RoboDK station: Conveying-Decanting-and-Material-Handling-with-Fanuc-R-2000iC-165F.rdk

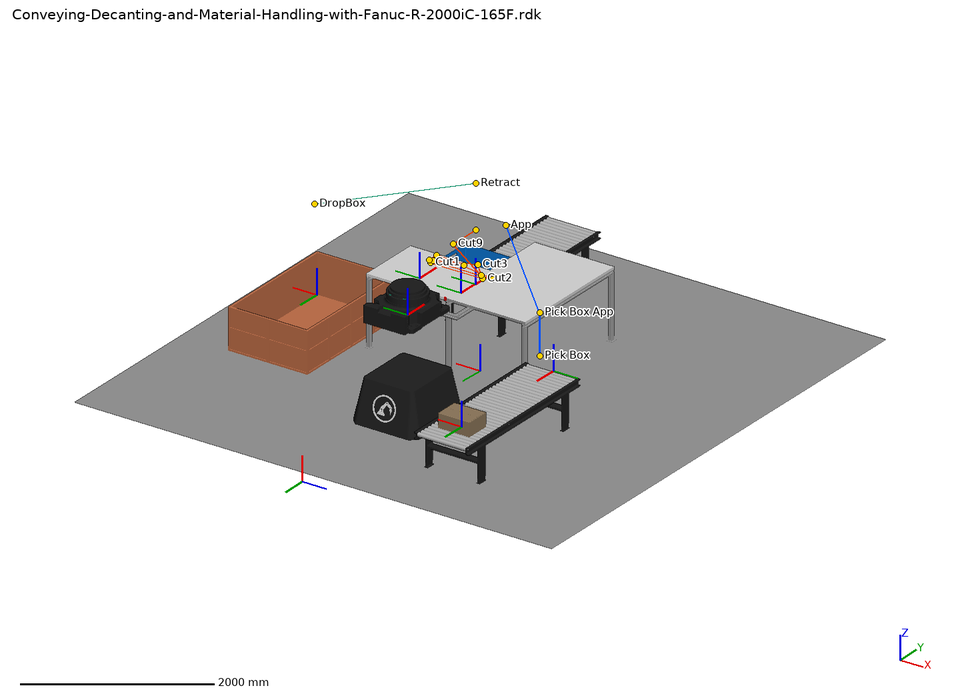
[picture v0: the station drawn from its stored meshes, robots at their saved joint values, targets as dots, program paths as lines]
Station Conveying, Decanting and Material Handling with Fanuc R-2000iC/165F (saved by RoboDK 5.9.2). Poses are relative to the parent item; angles as X-Y-Z fixed-axis rotations.
Station parameters (name, value as stored): TAGS, ['Decanting']
  - frame Roller Conveyor In Base at (1190, -380, 485) mm, rotated rx 0 ry 0 rz -90 deg
    - robot Roller Conveyor In: 1 axes
        modified DH rows (alpha deg, a mm, theta deg, d mm): 0, 0, 0, 0 linear
        base shift (0, 0, -485) mm, rotated rx 0 ry 90 rz 0 deg
        joint limits [-20000] to [20000]; home [0]; saved at [1400]
      - frame Conveyor In Ref at (230, -10, 5) mm, rotated rx 0 ry 0 rz -90 deg
        - frame BoxRef at (0, 0, 0) mm
          - object Decanting Box Bottom at (0, 0, 0) mm, size 400 x 300 x 6 mm, geometry from Decanting Box v4.step
          - object Decanting Box Top at (0, 0, 0) mm, size 400 x 300 x 166 mm, geometry from Decanting Box v4.step
          - object RoboDK_logo at (135, -20, 160) mm, rotated rx 0 ry 0 rz 90 deg, size 280 x 130 x 161.8 mm
          - object RoboDK_logo at (5, -20, 160) mm, rotated rx 0 ry 0 rz 90 deg, size 280 x 130 x 161.8 mm
          - object RoboDK_logo at (-125, -20, 160) mm, rotated rx 0 ry 0 rz 90 deg, size 280 x 130 x 161.8 mm
    - target Conv In 1 (Cartesian target) at (1400, 0, 0) mm; joints [1400, -18.458, 3.617, 0, -93.617, -148.241] of Roller Conveyor In
    - target Conv In 2 (Cartesian target) at (0, 0, 0) mm; joints [0, -18.458, 3.617, 0, -93.617, -148.241] of Roller Conveyor In
  - frame Roller Conveyor Out Base at (-640, 570, 485) mm, rotated rx 0 ry 0 rz 90 deg
    - robot Roller Conveyor Out: 1 axes
        modified DH rows (alpha deg, a mm, theta deg, d mm): 0, 0, 0, 0 linear
        base shift (0, 0, -485) mm, rotated rx 0 ry 90 rz 0 deg
        joint limits [-20000] to [20000]; home [0]; saved at [0]
      - frame Conveyor Out Ref at (250, -10, 0) mm
        - object Caisse Modulaire at (0, 0, 0) mm, size 460 x 580 x 300 mm, geometry from Caisse Modulaire v5.step
  - frame Gravity Base at (0, 0, 0) mm, rotated rx 0 ry 0 rz 180 deg
    - robot Gravity: 1 axes
        modified DH rows (alpha deg, a mm, theta deg, d mm): 0, 0, 0, 0 linear
        joint limits [0] to [900000]; home [0]; saved at [0]
      - frame GravityRef at (0, 3190, 0) mm
      - tool Gravity TCP, TCP at (0, 0, 0) mm
    - target BoxDrop1 (Cartesian target) at (0, 0, -355) mm, rotated rx 0 ry -90 rz 0 deg; joints [355, 40.194, -30.706, 0, -59.294, 73.523] of Gravity
    - target BoxDrop2 (Cartesian target) at (0, 0, -1505) mm, rotated rx 0 ry -90 rz 0 deg; joints [1505, 40.194, -30.706, 0, -59.294, 73.523] of Gravity
  - frame Fanuc R-2000iC/165F Base at (0, -1300, 1160) mm, rotated rx 0 ry 0 rz 90 deg
    - robot Fanuc R-2000iC/165F: 6 axes, payload 165 kg, reach 2655 mm, repeatability 0.2 mm, weight 1170 kg
        joint limits [-185, -56, -65, -360, -125, -360] to [185, 80, 245, 360, 125, 360]; home [0, 0, 0, 0, 0, 0]; saved at [5.758, -15.413, -35.804, 0, -54.196, -95.758]
      - tool Decanting gripper v3, TCP at (0, 0, 200) mm, size 405 x 200 x 270 mm, geometry from Decanting gripper v3.step
      - frame BoxOpening Base at (0, -148, 458) mm
        - robot BoxOpening: 1 axes
            modified DH rows (alpha deg, a mm, theta deg, d mm): 0, 0, 0, 0
            base shift (0, 0, 0) mm, rotated rx 0 ry 90 rz 0 deg
            joint limits [-360] to [360]; home [0]; saved at [0]
          - tool BoxOpeningTCP, TCP at (0, 0, 0) mm
    - object Pedestal H500mm (Type 2) at (0, 0, -1160) mm, rotated rx 0 ry 0 rz 90 deg, size 844.5 x 933.7 x 500 mm, geometry from Pedestal-H500mm-Type-2.sld
    - target Pick Box (Cartesian target) at (690, -1180, -415) mm, rotated rx -180 ry 0 rz -90 deg; joints [-59.683, 14.803, -63.072, 0, -26.928, -30.317] of Fanuc R-2000iC/165F
    - target Pick Box App (Cartesian target) at (690, -1180, 75) mm, rotated rx -180 ry 0 rz -90 deg; joints [-59.683, -5.784, -36.452, 0, -53.548, -30.317] of Fanuc R-2000iC/165F
    - target App (Cartesian target) at (1570, -140, 435) mm, rotated rx -180 ry 0 rz -90 deg; joints [-5.096, -0.842, -19.934, 0, -70.066, -84.904] of Fanuc R-2000iC/165F
    - frame Table at (1300, 0, -1160) mm, rotated rx 0 ry 0 rz 90 deg
      - object Decanting table assem at (-220, -1380, 485) mm, rotated rx 0 ry 0 rz -180 deg, size 2035.1 x 1855.1 x 855 mm, geometry from Decanting table assem v12.step
      - target Cut1 (Cartesian target) at (570, 70, 1106) mm, rotated rx 180 ry 0 rz -180 deg; joints [24.864, -2.283, -43.25, 0, -46.75, -114.864] of Fanuc R-2000iC/165F
      - target Cut2 (Cartesian target) at (-80, 70, 1106) mm, rotated rx 180 ry 0 rz 180 deg; joints [-3.721, -9.346, -42.545, 0, -47.455, -86.279] of Fanuc R-2000iC/165F
      - target Cut3 (Cartesian target) at (140, -170, 1106) mm, rotated rx 180 ry 0 rz -180 deg; joints [5.44, 4.103, -43.15, 0, -46.85, -95.44] of Fanuc R-2000iC/165F
      - target Cut4 (Cartesian target) at (570, 20, 1106) mm, rotated rx 180 ry 0 rz -90 deg; joints [24.004, 0.173, -43.295, 0, -46.705, -24.004] of Fanuc R-2000iC/165F
      - target Cut5 (Cartesian target) at (-170, 20, 1106) mm, rotated rx -180 ry 0 rz -90 deg; joints [-7.565, -5.895, -42.995, 0, -47.005, 7.565] of Fanuc R-2000iC/165F
      - target Cut6 (Cartesian target) at (620, -110, 1106) mm, rotated rx 180 ry 0 rz 0 deg; joints [23.736, 7.305, -42.836, 0, -47.164, 66.264] of Fanuc R-2000iC/165F
      - target Cut7 (Cartesian target) at (620, 20, 1106) mm, rotated rx 180 ry 0 rz 90 deg; joints [25.844, 1.287, -43.28, 0, -46.72, 154.156] of Fanuc R-2000iC/165F
      - target Cut8 (Cartesian target) at (-30, 20, 1106) mm, rotated rx 180 ry 0 rz 90 deg; joints [-1.343, -6.523, -42.928, 0, -47.072, 181.343] of Fanuc R-2000iC/165F
      - target Cut9 (Cartesian target) at (630, -420, 1106) mm, rotated rx -180 ry 0 rz 0 deg; joints [20.117, 21.228, -39.525, 0, -50.475, 69.883] of Fanuc R-2000iC/165F
      - target Cut10 (Cartesian target) at (630, -830, 1106) mm, rotated rx 180 ry 0 rz 0 deg; joints [16.477, 40.194, -30.706, 0, -59.294, 73.523] of Fanuc R-2000iC/165F
    - target Retract (Cartesian target) at (2130, 630, 476) mm, rotated rx -180 ry 0 rz 90 deg; joints [16.477, 34.546, -9.725, 0, -80.275, 73.523] of Fanuc R-2000iC/165F
    - target DropBox (Cartesian target) at (1120, 1950, 276) mm, rotated rx -180 ry 0 rz 90 deg; joints [60.129, 37.062, -17.345, 0, -72.655, 29.871] of Fanuc R-2000iC/165F
    - target Home (Cartesian target) at (1190, 120, 55) mm, rotated rx 180 ry 0 rz -90 deg; joints [5.758, -15.413, -35.804, 0, -54.196, -95.758] of Fanuc R-2000iC/165F
  - frame Container at (-2400, 500, 0) mm, rotated rx 0 ry 0 rz 180 deg
    - object Container at (0, 0, 0) mm, size 1000 x 1600 x 500 mm, geometry from Container.step
  - object Floor at (0, 0, 0) mm, rotated rx 0 ry 0 rz 180 deg, size 6000 x 6000 x 0 mm, geometry from Floor.sld
  - program Main (19 instructions, listed below)
  - folder Python
    - Python program OpenBox (listed below)
    - Python program MechnaismReset (listed below)
    - Python program ConveyorReset (listed below)
    - Python program SwitchRef_Box_to_convOut (listed below)
  - folder Programs
    - program Gravity_BoxDrop2 (3 instructions, listed below)
    - program CutBox (14 instructions, listed below)
    - program RecycleBox (7 instructions, listed below)
  - program Home (3 instructions, listed below)
  - program Conv In (2 instructions, listed below)
  - program Reset (4 instructions, listed below)
  - notes Description: <!DOCTYPE HTML PUBLIC "-//W3C//DTD HTML 4.0//EN" "http://www.w3.org/TR/REC-html40/strict.dtd">
<html><head><meta name="qrichtext" content="1" /><style type="text/css">
p, li { white-space: pre-wrap; }
</style></head><body style=" font-family:'MS Shell Dlg 2'; font-size:8.25pt; font-weight:400; font-style:normal;">
<p style=" margin-top:0px; margin-bottom:0px; margin-left:0px; margin-right:0px; -qt-block-indent:0; text-indent:0px;">This example demonstrates a box emptying and sorting application using an industrial 6-axis Fanuc R-2000iC/165F robot equipped with a vacuum gripper. The robot picks a closed box from a roller conveyor and opens its bottom by sliding it across a stationary knife mounted on a flat table. It then pushes the opened box toward a bin, allowing the contents to fall out. After emptying, the robot discards the empty box into a designated container.</p></body></html>
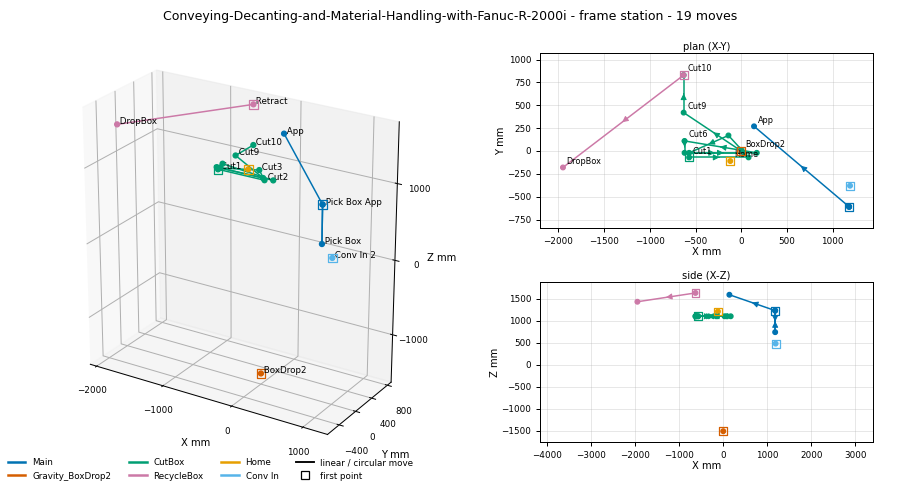
[picture p0: tool path of Conveying-Decanting-and-Material-Handling-with-Fanuc-R-2000iC-165F.rdk in frame station, 19 of 19 moves have a stored position in this frame; points joined in program order, loops and branches not executed]

--- program Main (robot Fanuc R-2000iC/165F) ---
  Call Reset
  Set Ref.: Fanuc R-2000iC/165F Base
  Set Tool: Decanting gripper v3
  Call Home
  Call Conv In
  MoveJ (Pick Box App)
  MoveL (Pick Box)
  Attach to Decanting gripper v3
  Attach to Decanting gripper v3
  Attach to Decanting gripper v3
  Attach to Decanting gripper v3
  Attach to Decanting gripper v3
  MoveL (Pick Box App)
  MoveL (App)
  Call CutBox
  Call OpenBox
  Call SwitchRef_Box_to_convOut
  Call RecycleBox
  Call Home

--- Python program OpenBox ---
# Type help("robodk.robolink") or help("robodk.robomath") for more information
# Press F5 to run the script
# Documentation: https://robodk.com/doc/en/RoboDK-API.html
# Reference:     https://robodk.com/doc/en/PythonAPI/robodk.html
# Note: It is not required to keep a copy of this file, your Python script is saved with your RDK project

# You can also use the new version of the API:
from robodk import robolink    # RoboDK API
from robodk import robomath    # Robot toolbox
import time
RDK = robolink.Robolink()

#----- Constant -----

MECHANISM_NAME1 = 'BoxOpening'
MECHANISM_NAME2 = 'Gravity'
PART_TRAVEL_MM = 0
Target1 = RDK.Item("BoxDrop1")

#Declaration of the frames
frame1 = RDK.Item('Decanting gripper v3')
frame2 = RDK.Item('BoxOpeningTCP')

item1 = RDK.Item("Decanting Box Bottom")
item2 = RDK.Item("RoboDK_logo")

gravityframe = RDK.Item("GravityRef")

#Declaration of the child frames
obj_list1 = frame1.Childs()
obj_list2 = frame2.Childs()

mechanism1 = RDK.Item(MECHANISM_NAME1)
mechanism2 = RDK.Item(MECHANISM_NAME2)

if mechanism1.Valid():
  mechanism1.MoveJ([0])

#open box
for item in obj_list1:
  if item.Name() == item1.Name():
      item.setParentStatic(frame2)

if mechanism1.Valid():
  mechanism1.MoveJ([90])

for item in obj_list2:
    item.setParentStatic(frame1)

#drop box
for item in obj_list1:
  if item.Name() == item1.Name():
    item.setParentStatic(frame2)

#Gravity
for item in obj_list1:
  if item.Name() == item2.Name():
    item.setParentStatic(gravityframe)

if mechanism2.Valid():
  mechanism2.setJoints([0])
  mechanism2.MoveL(Target1)

--- Python program MechnaismReset ---
# Type help("robodk.robolink") or help("robodk.robomath") for more information
# Press F5 to run the script
# Documentation: https://robodk.com/doc/en/RoboDK-API.html
# Reference:     https://robodk.com/doc/en/PythonAPI/robodk.html
# Note: It is not required to keep a copy of this file, your Python script is saved with your RDK project

# You can also use the new version of the API:
from robodk import robolink    # RoboDK API
from robodk import robomath    # Robot toolbox
RDK = robolink.Robolink()

#----- Constant -----

MECHANISM_NAME1 = 'BoxOpening'
MECHANISM_NAME2 = 'Gravity'

mechanism1 = RDK.Item(MECHANISM_NAME1)
mechanism2 = RDK.Item(MECHANISM_NAME2)

if mechanism1.Valid():
  mechanism1.setJoints([0])

if mechanism2.Valid():
  mechanism2.setJoints([0])

--- Python program ConveyorReset ---
# Type help("robodk.robolink") or help("robodk.robomath") for more information
# Press F5 to run the script
# Documentation: https://robodk.com/doc/en/RoboDK-API.html
# Reference:     https://robodk.com/doc/en/PythonAPI/robodk.html
# Note: It is not required to keep a copy of this file, your Python script is saved with your RDK project

# You can also use the new version of the API:
from robodk import robolink    # RoboDK API
from robodk import robomath    # Robot toolbox
RDK = robolink.Robolink()

#----- Constant -----
MECHANISM_NAME1 = 'Roller Conveyor In'#Name of the conveyor mechanism
MECHANISM_NAME2 = 'Roller Conveyor Out'#Name of the conveyor mechanism
MECHANISM_NAME3 = 'Gravity'#Name of the conveyor mechanism
PART_TRAVEL_MM = 0 #Travel for each box

mechanism1 = RDK.Item(MECHANISM_NAME1)
if mechanism1.Valid():
    mechanism1.setJoints([1400.00])

mechanism2 = RDK.Item(MECHANISM_NAME2)
if mechanism2.Valid():
    mechanism2.setJoints([0])


mechanism3 = RDK.Item(MECHANISM_NAME3)
if mechanism3.Valid():
    mechanism3.setJoints([0])

--- Python program SwitchRef_Box_to_convOut ---
# Type help("robodk.robolink") or help("robodk.robomath") for more information
# Press F5 to run the script
# Documentation: https://robodk.com/doc/en/RoboDK-API.html
# Reference:     https://robodk.com/doc/en/PythonAPI/robodk.html
# Note: It is not required to keep a copy of this file, your Python script is saved with your RDK project

# You can also use the new version of the API:
from robodk import robolink    # RoboDK API
from robodk import robomath    # Robot toolbox
import time
RDK = robolink.Robolink()

#----- Constant -----
Target1 = RDK.Item("BoxDrop1")

#Declaration of the frames
frame3 = RDK.Item("Conveyor Out Ref")

item1 = RDK.Item("Decanting Box Bottom")
item2 = RDK.Item("RoboDK_logo")

gravityframe = RDK.Item("GravityRef")

#Declaration of the child frames
obj_list4 = gravityframe.Childs()

#Switch to conveyor ref
for item in obj_list4:
    item.setParentStatic(frame3)

--- program Gravity_BoxDrop2 (robot Gravity) ---
  Set Ref.: Gravity Base
  Set Tool: Gravity TCP
  MoveL (BoxDrop2)

--- program CutBox (robot Fanuc R-2000iC/165F) ---
  Set Ref.: Table
  Set Tool: Decanting gripper v3
  Set speed (200.0 mm/s)
  MoveL (Cut1)
  MoveL (Cut2)
  MoveL (Cut3)
  MoveL (Cut4)
  MoveL (Cut5)
  MoveL (Cut6)
  MoveL (Cut7)
  MoveL (Cut8)
  MoveL (Cut9)
  MoveL (Cut10)
  Set speed (600.0 mm/s)

--- program RecycleBox (robot Fanuc R-2000iC/165F) ---
  Set Ref.: Fanuc R-2000iC/165F Base
  Set Tool: Decanting gripper v3
  MoveL (Retract)
  MoveL (DropBox)
  Detach from Decanting gripper v3
  Detach from BoxOpeningTCP
  Call Gravity_BoxDrop2

--- program Home (robot Fanuc R-2000iC/165F) ---
  Set Ref.: Fanuc R-2000iC/165F Base
  Set Tool: Decanting gripper v3
  MoveJ (Home)

--- program Conv In (robot Roller Conveyor In) ---
  Set Ref.: Roller Conveyor In Base
  MoveJ (Conv In 2)

--- program Reset (robot Fanuc R-2000iC/165F) ---
  Call ConveyorReset
  Replace objects
  Call MechnaismReset
  Call Home
